PROGRAM PRG_Logging

VAR
    fbLogger : FB_Logger;
END_VAR

fbLogger();

METHOD PUBLIC M_SysLog : HRESULT
VAR_INPUT
END_VAR
END_METHOD

END_PROGRAM

(* stored: Version 1.1.0.1
   POU PRG_Logging: Id {62911cf1-27d8-438e-b3ad-1711808e3e53}, SpecialFunc None
   Method M_SysLog: Id {2c8e93f3-e53d-4e3e-9d2d-9ea4f5579afe} *)
